PROGRAM PIST_CYCLE
VAR
	bFirstRun:BOOL:=FALSE;
	counter :INT;
END_VAR


//IF NOT bFirstRun THEN
//	FOR counter:=1 TO iNUMBER_OF_PISTONS BY 1 DO
//		fbPist[counter].bInit:=1;
//	END_FOR;
//bFirstRun:=TRUE;
//END_IF
 

grp1();

ACTION grp1:
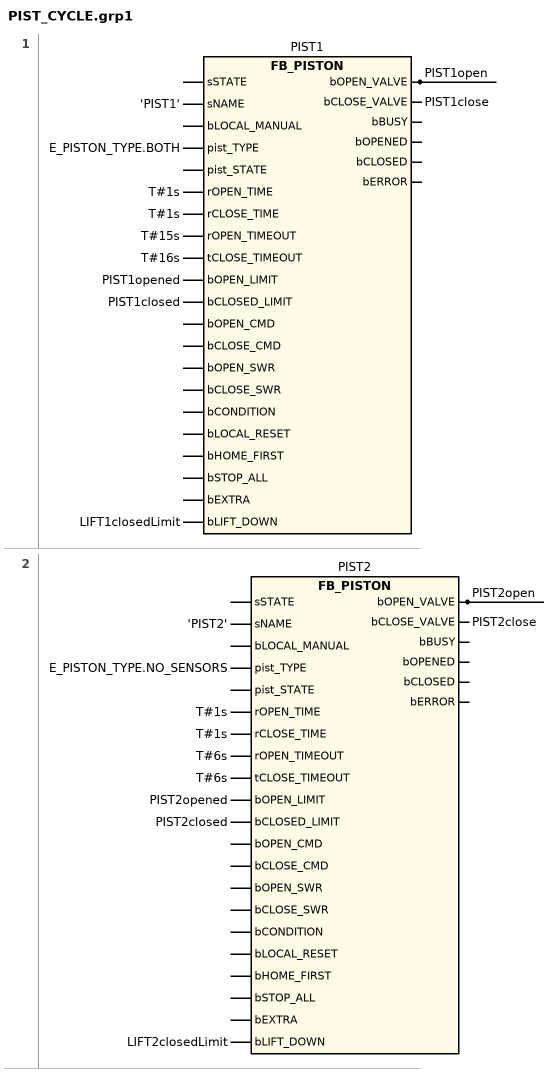
// NETWORK 1
PIST1(
    sNAME := 'PIST1',
    pist_TYPE := E_PISTON_TYPE.BOTH,
    rOPEN_TIME := T#1s,
    rCLOSE_TIME := T#1s,
    rOPEN_TIMEOUT := T#15s,
    tCLOSE_TIMEOUT := T#16s,
    bOPEN_LIMIT := PIST1opened,
    bCLOSED_LIMIT := PIST1closed,
    bLIFT_DOWN := LIFT1closedLimit,
    bOPEN_VALVE => PIST1open,
    bCLOSE_VALVE => PIST1close); // FB_PISTON

// NETWORK 2
PIST2(
    sNAME := 'PIST2',
    pist_TYPE := E_PISTON_TYPE.NO_SENSORS,
    rOPEN_TIME := T#1s,
    rCLOSE_TIME := T#1s,
    rOPEN_TIMEOUT := T#6s,
    tCLOSE_TIMEOUT := T#6s,
    bOPEN_LIMIT := PIST2opened,
    bCLOSED_LIMIT := PIST2closed,
    bLIFT_DOWN := LIFT2closedLimit,
    bOPEN_VALVE => PIST2open,
    bCLOSE_VALVE => PIST2close); // FB_PISTON
END_ACTION

END_PROGRAM

(* stored: Version 1.1.0.1, ProductVersion 3.1.4024.12
   POU PIST_CYCLE: Id {b09e4efb-d7ec-45c6-bc50-8222237b347f}, SpecialFunc None
   Action grp1: Id {b6db8f46-a5cd-4841-b2f4-af5cb236d344} *)
